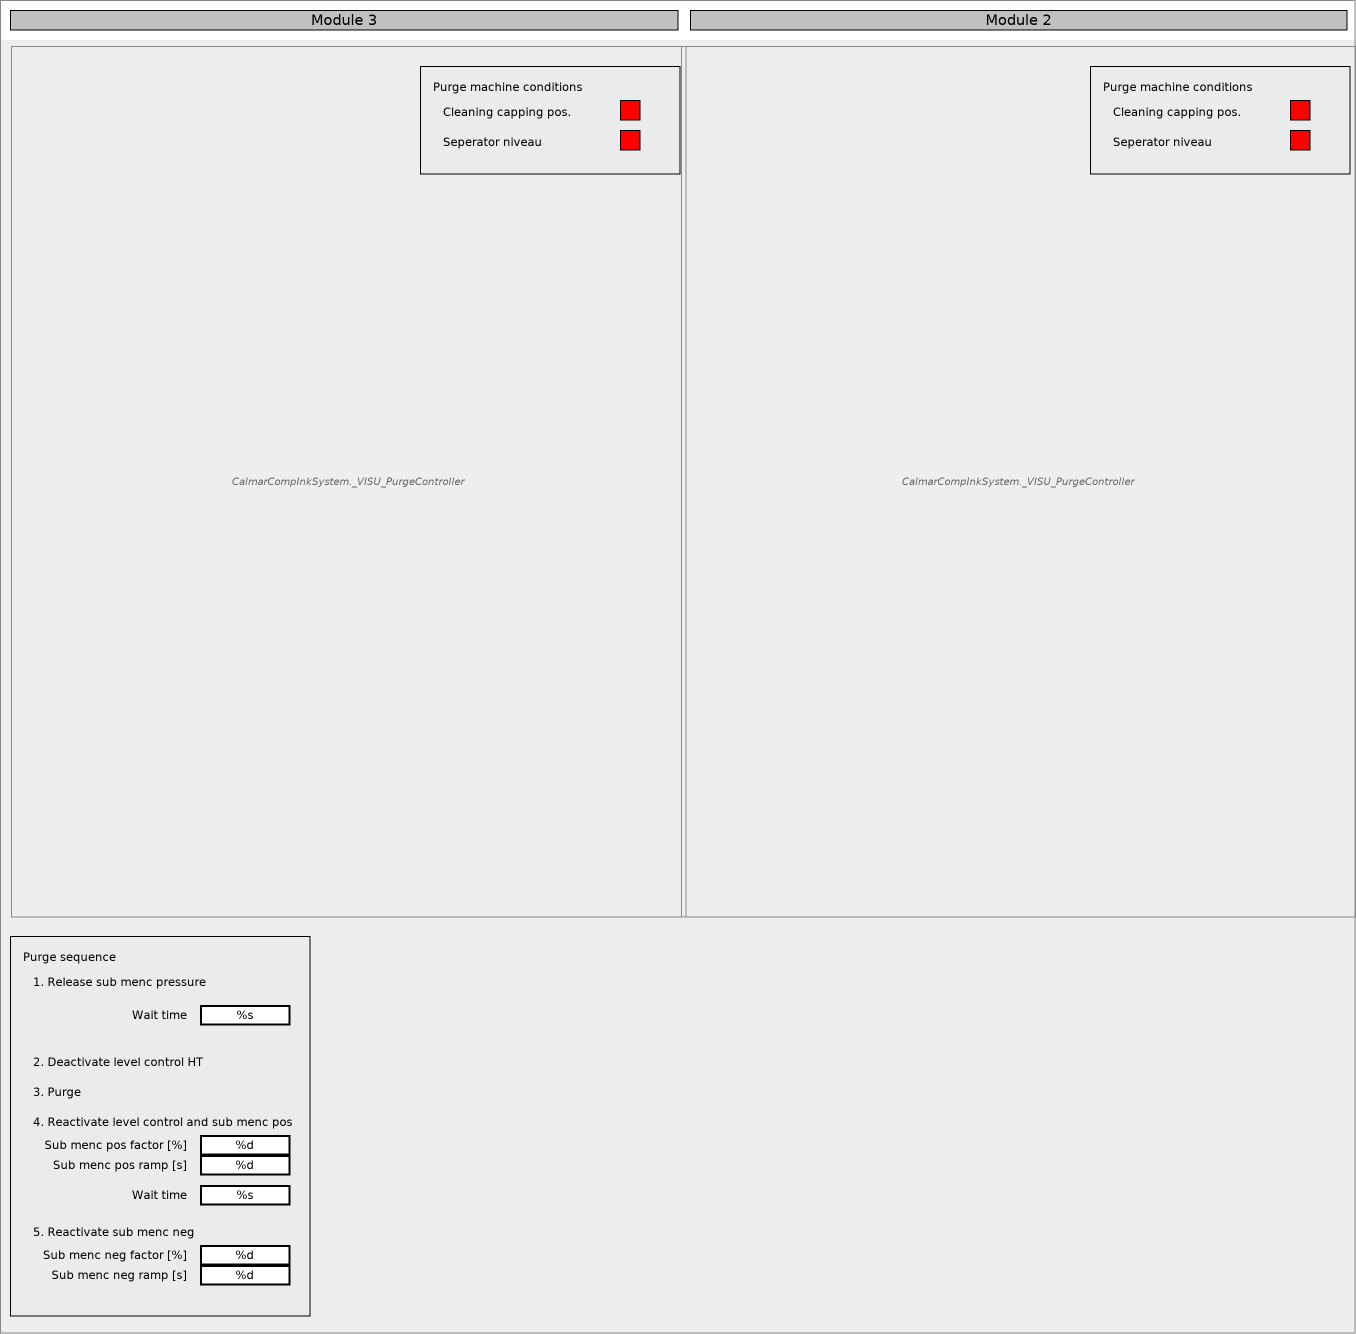
VISUALIZATION VISU_PURGE  // 1356x1334
    Rectangle (0,40 1356x1294)
    Frame (11,46 675x871)
        shows CalmarCompInkSystem._VISU_PurgeController(m_Inst_Fb := PRG_INK.fb_PurgeController[2])
    Rectangle (10,936 300x380), invisible if: (bCIk_PURGE_CONTR_SEQUENCE[1] = FALSE) and (bCIk_PURGE_CONTR_SEQUENCE[2] = FALSE)
    Rectangle (20,947 150x20), "Purge sequence", invisible if: (bCIk_PURGE_CONTR_SEQUENCE[1] = FALSE) and (bCIk_PURGE_CONTR_SEQUENCE[2] = FALSE)
    Rectangle (30,972 204x20), "1. Release sub menc pressure", invisible if: (bCIk_PURGE_CONTR_SEQUENCE[1] = FALSE) and (bCIk_PURGE_CONTR_SEQUENCE[2] = FALSE)
    Rectangle (60,1005 130x20), "Wait time", invisible if: (bCIk_PURGE_CONTR_SEQUENCE[1] = FALSE) and (bCIk_PURGE_CONTR_SEQUENCE[2] = FALSE)
    Rectangle (200,1005 90x20), "%s", text variable: PRG_INK.fb_PurgeController[1].tR_ReleaseTime, invisible if: (bCIk_PURGE_CONTR_SEQUENCE[1] = FALSE) and (bCIk_PURGE_CONTR_SEQUENCE[2] = FALSE)
        OnMouseDown: write the text variable via Edit
    Rectangle (30,1052 204x20), "2. Deactivate level control HT", invisible if: (bCIk_PURGE_CONTR_SEQUENCE[1] = FALSE) and (bCIk_PURGE_CONTR_SEQUENCE[2] = FALSE)
    Rectangle (30,1082 204x20), "3. Purge", invisible if: (bCIk_PURGE_CONTR_SEQUENCE[1] = FALSE) and (bCIk_PURGE_CONTR_SEQUENCE[2] = FALSE)
    Rectangle (30,1112 275x20), "4. Reactivate level control and sub menc pos", invisible if: (bCIk_PURGE_CONTR_SEQUENCE[1] = FALSE) and (bCIk_PURGE_CONTR_SEQUENCE[2] = FALSE)
    Rectangle (40,1135 150x20), "Sub menc pos factor [%]", invisible if: (bCIk_PURGE_CONTR_SEQUENCE[1] = FALSE) and (bCIk_PURGE_CONTR_SEQUENCE[2] = FALSE)
    Rectangle (200,1135 90x20), "%d", text variable: PRG_INK.fb_PurgeController[1].iR_SubMencPosFactor, invisible if: (bCIk_PURGE_CONTR_SEQUENCE[1] = FALSE) and (bCIk_PURGE_CONTR_SEQUENCE[2] = FALSE)
        OnMouseDown: write the text variable via Edit, min 1, max 100
    Rectangle (30,1222 250x20), "5. Reactivate sub menc neg", invisible if: (bCIk_PURGE_CONTR_SEQUENCE[1] = FALSE) and (bCIk_PURGE_CONTR_SEQUENCE[2] = FALSE)
    Rectangle (60,1185 130x20), "Wait time", invisible if: (bCIk_PURGE_CONTR_SEQUENCE[1] = FALSE) and (bCIk_PURGE_CONTR_SEQUENCE[2] = FALSE)
    Rectangle (200,1185 90x20), "%s", text variable: PRG_INK.fb_PurgeController[1].tR_SubMencReactivateTime, invisible if: (bCIk_PURGE_CONTR_SEQUENCE[1] = FALSE) and (bCIk_PURGE_CONTR_SEQUENCE[2] = FALSE)
        OnMouseDown: write the text variable via Edit
    Rectangle (40,1155 150x20), "Sub menc pos ramp [s]", invisible if: (bCIk_PURGE_CONTR_SEQUENCE[1] = FALSE) and (bCIk_PURGE_CONTR_SEQUENCE[2] = FALSE)
    Rectangle (200,1155 90x20), "%d", text variable: PRG_INK.fb_PurgeController[1].tR_SubMencPosRampTime, invisible if: (bCIk_PURGE_CONTR_SEQUENCE[1] = FALSE) and (bCIk_PURGE_CONTR_SEQUENCE[2] = FALSE)
        OnMouseDown: write the text variable via Edit
    Rectangle (40,1245 150x20), "Sub menc neg factor [%]", invisible if: (bCIk_PURGE_CONTR_SEQUENCE[1] = FALSE) and (bCIk_PURGE_CONTR_SEQUENCE[2] = FALSE)
    Rectangle (200,1245 90x20), "%d", text variable: PRG_INK.fb_PurgeController[1].iR_SubMencNegFactor, invisible if: (bCIk_PURGE_CONTR_SEQUENCE[1] = FALSE) and (bCIk_PURGE_CONTR_SEQUENCE[2] = FALSE)
        OnMouseDown: write the text variable via Edit, min 1, max 100
    Rectangle (40,1265 150x20), "Sub menc neg ramp [s]", invisible if: (bCIk_PURGE_CONTR_SEQUENCE[1] = FALSE) and (bCIk_PURGE_CONTR_SEQUENCE[2] = FALSE)
    Rectangle (200,1265 90x20), "%d", text variable: PRG_INK.fb_PurgeController[1].tR_SubMencNegRampTime, invisible if: (bCIk_PURGE_CONTR_SEQUENCE[1] = FALSE) and (bCIk_PURGE_CONTR_SEQUENCE[2] = FALSE)
        OnMouseDown: write the text variable via Edit
    Rectangle (420,66 260x108)
    Rectangle (430,77 203x20), "Purge machine conditions"
    Rectangle (440,102 148x20), "Cleaning capping pos."
    RoundedRectangle (620,100 20x20), colour toggle: PRG_MACHINE.fb_CleaningCU[2].pInPosCappingClean
    Rectangle (440,132 148x20), "Seperator niveau"
    RoundedRectangle (620,130 20x20), colour toggle: PRG_MACHINE.bIKp_SeparatorNiveau_Ok[2]
    Frame (681,46 675x871)
        shows CalmarCompInkSystem._VISU_PurgeController(m_Inst_Fb := PRG_INK.fb_PurgeController[1])
    Rectangle (1090,66 260x108)
    Rectangle (1100,77 203x20), "Purge machine conditions"
    Rectangle (1110,102 148x20), "Cleaning capping pos."
    RoundedRectangle (1290,100 20x20), colour toggle: PRG_MACHINE.fb_CleaningCU[1].pInPosCappingClean
    Rectangle (1110,132 148x20), "Seperator niveau"
    RoundedRectangle (1290,130 20x20), colour toggle: PRG_MACHINE.bIKp_SeparatorNiveau_Ok[1]
    Rectangle (10,10 668x20), "Module 3"
    Rectangle (690,10 657x20), "Module 2"
END_VISUALIZATION

(* stored: Version 1.1.0.1, ProductVersion 3.1.4024.11
   Visu VISU_PURGE: Id {26cea0c8-0a15-4453-963c-beaa616d340a} *)
